TYPE STMStatus :
STRUCT
	readyToEnable : BOOL;
	ready : BOOL;
	warning : BOOL;
	error : BOOL;
	movingPositive : BOOL;
	movingNegative : BOOL;
	txPDOToggle : BOOL;
END_STRUCT
END_TYPE

(* stored: Version 1.1.0.1, ProductVersion 3.1.4024.9
   DUT STMStatus: Id {66f75789-f59b-45e6-9cf0-983aa11de110} *)
